PROGRAM P4_05_DIskSize
VAR
	fbSize				:FB_PythonScript;
END_VAR

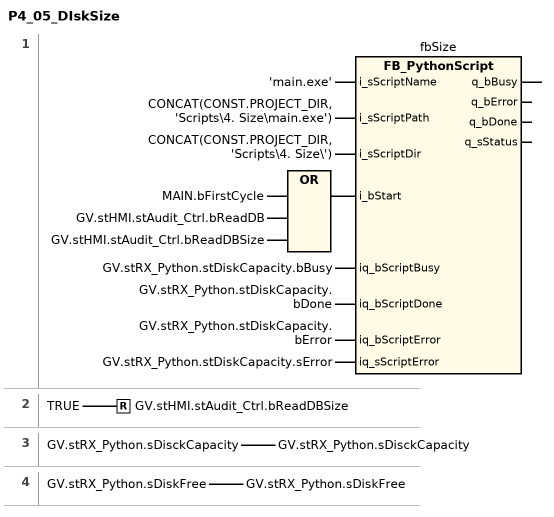
// NETWORK 1
fbSize(
    i_sScriptName := 'main.exe',
    i_sScriptPath := CONCAT(CONST.PROJECT_DIR,'Scripts\4. Size\main.exe'),
    i_sScriptDir := CONCAT(CONST.PROJECT_DIR,'Scripts\4. Size\'),
    i_bStart := MAIN.bFirstCycle OR GV.stHMI.stAudit_Ctrl.bReadDB OR GV.stHMI.stAudit_Ctrl.bReadDBSize,
    iq_bScriptBusy := GV.stRX_Python.stDiskCapacity.bBusy,
    iq_bScriptDone := GV.stRX_Python.stDiskCapacity.bDone,
    iq_bScriptError := GV.stRX_Python.stDiskCapacity.bError,
    iq_sScriptError := GV.stRX_Python.stDiskCapacity.sError); // FB_PythonScript

// NETWORK 2
GV.stHMI.stAudit_Ctrl.bReadDBSize R= TRUE;

// NETWORK 3
GV.stRX_Python.sDisckCapacity := GV.stRX_Python.sDisckCapacity;

// NETWORK 4
GV.stRX_Python.sDiskFree := GV.stRX_Python.sDiskFree;

END_PROGRAM

(* stored: Version 1.1.0.1
   POU P4_05_DIskSize: Id {37c73627-27c3-4fae-9810-f82ba81eb48e}, SpecialFunc None *)
